PROGRAM P_Clock
VAR
	
	fbClock : FB_Clock;
	fbMotionClock : FB_Clock;
	fbDriveOut : FB_Clock;
	
END_VAR


fbClock(
	bStartEnable := G_HMI.bstepp_button,
	
	fTime => G_OPC.fTime
);

fbMotionClock(
	bStartEnable := G_Enables.bSineMotion AND G_Enables.bHoldButton AND G_Enables.bAuto, // AND G_HMI.bstepp_button AND G_Enables.bHoldButton,
	
	fTime => G_OPC.fMotionTime
);

fbDriveOut(
	bStartEnable := G_Truck.bDriveOut AND NOT(G_HMI.bstepp_button),
	
	fTime => G_Truck.fDriveOutTime
);

END_PROGRAM

(* stored: Version 1.1.0.1
   POU P_Clock: Id {3607f292-5366-4b7c-810f-569374c051f5}, SpecialFunc None *)
